(* IEC 61131-3 sources: AXOpen/src/components.cognex.vision/app/SystemConstants, 6 files *)

(* ---- plc_line_1518_HwIdentifiers.st ---- *)
CONFIGURATION HardwareIDs
    VAR_GLOBAL CONSTANT
        dm_280_HwID : UINT := UINT#299;
        dm_280_Acquisition_Control_Acquisition_Control_HwID : UINT := UINT#309;
        dm_280_Acquisition_Status_Acquisition_Status_HwID : UINT := UINT#306;
        dm_280_Rack_HwID : UINT := UINT#301;
        dm_280_Result_Data_128_bytes_Result_Data___128_bytes_HwID : UINT := UINT#303;
        dm_280_Results_Control_Results_Control_HwID : UINT := UINT#308;
        dm_280_Results_Status_Results_Status_HwID : UINT := UINT#305;
        dm_280_Soft_Event_Control_Soft_Event_Control_HwID : UINT := UINT#307;
        dm_280_User_Data_128_bytes_User_Data___128_bytes_HwID : UINT := UINT#304;
        dm_280_dm_280_HwID : UINT := UINT#302;
        dm_280_dm_280_DataMan_280_CC_B_HwID : UINT := UINT#310;
        dm_280_dm_280_profinet_HwID : UINT := UINT#298;
        dm_280_dm_280_profinet_Port_1_HwID : UINT := UINT#300;
        dm_300_HwID : UINT := UINT#286;
        dm_300_Acquisition_Control_Acquisition_Control_HwID : UINT := UINT#296;
        dm_300_Acquisition_Status_Acquisition_Status_HwID : UINT := UINT#293;
        dm_300_Rack_HwID : UINT := UINT#288;
        dm_300_Result_Data_64_bytes_Result_Data___64_bytes_HwID : UINT := UINT#290;
        dm_300_Results_Control_Results_Control_HwID : UINT := UINT#295;
        dm_300_Results_Status_Results_Status_HwID : UINT := UINT#292;
        dm_300_Soft_Event_Control_Soft_Event_Control_HwID : UINT := UINT#294;
        dm_300_User_Data_64_bytes_User_Data___64_bytes_HwID : UINT := UINT#291;
        dm_300_dm_300_HwID : UINT := UINT#289;
        dm_300_dm_300_DataMan_300_HwID : UINT := UINT#297;
        dm_300_dm_300_profinet_HwID : UINT := UINT#285;
        dm_300_dm_300_profinet_Port_1_HwID : UINT := UINT#287;
        is2800_HwID : UINT := UINT#258;
        is2800_Acquisition_Control_Acquisition_Control_HwID : UINT := UINT#269;
        is2800_Acquisition_Status_Acquisition_Status_HwID : UINT := UINT#264;
        is2800_Command_Control_Command_Control_HwID : UINT := UINT#266;
        is2800_Inspection_Control_Inspection_Control_HwID : UINT := UINT#268;
        is2800_Inspection_Status_Inspection_Status_HwID : UINT := UINT#265;
        is2800_Rack_HwID : UINT := UINT#260;
        is2800_Result_Data_64_bytes_Results___64_bytes_HwID : UINT := UINT#262;
        is2800_SoftEvent_Control_ExternalEvent_Control_HwID : UINT := UINT#267;
        is2800_User_Data_64_bytes_User_Data___64_bytes_HwID : UINT := UINT#263;
        is2800_is2800_HwID : UINT := UINT#261;
        is2800_is2800_In_Sight_IS28XX_CC_B_HwID : UINT := UINT#270;
        is2800_is2800_profinet_HwID : UINT := UINT#257;
        is2800_is2800_profinet_Port_1_HwID : UINT := UINT#259;
        is7600_HwID : UINT := UINT#272;
        is7600_Acquisition_Control_Acquisition_Control_HwID : UINT := UINT#283;
        is7600_Acquisition_Status_Acquisition_Status_HwID : UINT := UINT#279;
        is7600_Command_Control_Command_Control_HwID : UINT := UINT#280;
        is7600_Inspection_Control_Inspection_Control_HwID : UINT := UINT#282;
        is7600_Inspection_Status_Inspection_Status_HwID : UINT := UINT#278;
        is7600_Rack_HwID : UINT := UINT#274;
        is7600_Result_Data_64_bytes_Results___64_bytes_HwID : UINT := UINT#276;
        is7600_SoftEvent_Control_SoftEvent_Control_HwID : UINT := UINT#281;
        is7600_User_Data_64_bytes_User_Data___64_bytes_HwID : UINT := UINT#277;
        is7600_is7600_HwID : UINT := UINT#275;
        is7600_is7600_In_Sight_IS79XX_IS75XX_CC_B_HwID : UINT := UINT#284;
        is7600_is7600_profinet_HwID : UINT := UINT#271;
        is7600_is7600_profinet_Port_1_HwID : UINT := UINT#273;
        plc_line_1518_HwID : UINT := UINT#32;
        plc_line_1518_Rail_0_HwID : UINT := UINT#311;
        plc_line_1518_plc_line_1518_HwID : UINT := UINT#48;
        plc_line_1518_plc_line_1518_CPU_display_1_HwID : UINT := UINT#54;
        plc_line_1518_plc_line_1518_Card_reader_writer_1_HwID : UINT := UINT#51;
        plc_line_1518_plc_line_1518_OPC_UA_1_HwID : UINT := UINT#117;
        plc_line_1518_plc_line_1518_Virtual_communication_interface_HwID : UINT := UINT#135;
        plc_line_1518_plc_line_1518_profinet_x1_HwID : UINT := UINT#64;
        plc_line_1518_plc_line_1518_profinet_x1_Port_1_HwID : UINT := UINT#65;
        plc_line_1518_plc_line_1518_profinet_x1_Port_2_HwID : UINT := UINT#66;
        plc_line_1518_plc_line_1518_profinet_x2_HwID : UINT := UINT#72;
        plc_line_1518_plc_line_1518_profinet_x2_Port_3_HwID : UINT := UINT#73;
        plc_line_1518_plc_line_1518_profinet_x2_Port_4_HwID : UINT := UINT#74;
        plc_line_1518_plc_line_1518_profinet_x3_HwID : UINT := UINT#120;
        plc_line_1518_plc_line_1518_profinet_x3_Port_5_HwID : UINT := UINT#121;
        profinet_plc_line_1518_HwID : UINT := UINT#256;

    END_VAR
END_CONFIGURATION

(* ---- plc_line_1518_IoAddresses.st ---- *)
CONFIGURATION IoAddresses
    VAR_GLOBAL
        dm_280_Acquisition_Control_OutputAddress AT %QB343: BYTE;
        dm_280_Acquisition_Status_InputAddress_0 AT %IB373: BYTE;
        dm_280_Acquisition_Status_InputAddress_1 AT %IB374: BYTE;
        dm_280_Acquisition_Status_InputAddress_2 AT %IB375: BYTE;
        dm_280_Result_Data_128_bytes_InputAddress_0 AT %IL236: LWORD;
        dm_280_Result_Data_128_bytes_InputAddress_1 AT %IL244: LWORD;
        dm_280_Result_Data_128_bytes_InputAddress_2 AT %IL252: LWORD;
        dm_280_Result_Data_128_bytes_InputAddress_3 AT %IL260: LWORD;
        dm_280_Result_Data_128_bytes_InputAddress_4 AT %IL268: LWORD;
        dm_280_Result_Data_128_bytes_InputAddress_5 AT %IL276: LWORD;
        dm_280_Result_Data_128_bytes_InputAddress_6 AT %IL284: LWORD;
        dm_280_Result_Data_128_bytes_InputAddress_7 AT %IL292: LWORD;
        dm_280_Result_Data_128_bytes_InputAddress_8 AT %IL300: LWORD;
        dm_280_Result_Data_128_bytes_InputAddress_9 AT %IL308: LWORD;
        dm_280_Result_Data_128_bytes_InputAddress_10 AT %IL316: LWORD;
        dm_280_Result_Data_128_bytes_InputAddress_11 AT %IL324: LWORD;
        dm_280_Result_Data_128_bytes_InputAddress_12 AT %IL332: LWORD;
        dm_280_Result_Data_128_bytes_InputAddress_13 AT %IL340: LWORD;
        dm_280_Result_Data_128_bytes_InputAddress_14 AT %IL348: LWORD;
        dm_280_Result_Data_128_bytes_InputAddress_15 AT %IL356: LWORD;
        dm_280_Result_Data_128_bytes_InputAddress_16 AT %IL364: LWORD;
        dm_280_Results_Control_OutputAddress AT %QB342: BYTE;
        dm_280_Results_Status_InputAddress AT %IB372: BYTE;
        dm_280_Soft_Event_Control_InputAddress AT %IB376: BYTE;
        dm_280_Soft_Event_Control_OutputAddress AT %QB341: BYTE;
        dm_280_User_Data_128_bytes_OutputAddress_0 AT %QD209: DWORD;
        dm_280_User_Data_128_bytes_OutputAddress_1 AT %QD213: DWORD;
        dm_280_User_Data_128_bytes_OutputAddress_2 AT %QD217: DWORD;
        dm_280_User_Data_128_bytes_OutputAddress_3 AT %QD221: DWORD;
        dm_280_User_Data_128_bytes_OutputAddress_4 AT %QD225: DWORD;
        dm_280_User_Data_128_bytes_OutputAddress_5 AT %QD229: DWORD;
        dm_280_User_Data_128_bytes_OutputAddress_6 AT %QD233: DWORD;
        dm_280_User_Data_128_bytes_OutputAddress_7 AT %QD237: DWORD;
        dm_280_User_Data_128_bytes_OutputAddress_8 AT %QD241: DWORD;
        dm_280_User_Data_128_bytes_OutputAddress_9 AT %QD245: DWORD;
        dm_280_User_Data_128_bytes_OutputAddress_10 AT %QD249: DWORD;
        dm_280_User_Data_128_bytes_OutputAddress_11 AT %QD253: DWORD;
        dm_280_User_Data_128_bytes_OutputAddress_12 AT %QD257: DWORD;
        dm_280_User_Data_128_bytes_OutputAddress_13 AT %QD261: DWORD;
        dm_280_User_Data_128_bytes_OutputAddress_14 AT %QD265: DWORD;
        dm_280_User_Data_128_bytes_OutputAddress_15 AT %QD269: DWORD;
        dm_280_User_Data_128_bytes_OutputAddress_16 AT %QD273: DWORD;
        dm_280_User_Data_128_bytes_OutputAddress_17 AT %QD277: DWORD;
        dm_280_User_Data_128_bytes_OutputAddress_18 AT %QD281: DWORD;
        dm_280_User_Data_128_bytes_OutputAddress_19 AT %QD285: DWORD;
        dm_280_User_Data_128_bytes_OutputAddress_20 AT %QD289: DWORD;
        dm_280_User_Data_128_bytes_OutputAddress_21 AT %QD293: DWORD;
        dm_280_User_Data_128_bytes_OutputAddress_22 AT %QD297: DWORD;
        dm_280_User_Data_128_bytes_OutputAddress_23 AT %QD301: DWORD;
        dm_280_User_Data_128_bytes_OutputAddress_24 AT %QD305: DWORD;
        dm_280_User_Data_128_bytes_OutputAddress_25 AT %QD309: DWORD;
        dm_280_User_Data_128_bytes_OutputAddress_26 AT %QD313: DWORD;
        dm_280_User_Data_128_bytes_OutputAddress_27 AT %QD317: DWORD;
        dm_280_User_Data_128_bytes_OutputAddress_28 AT %QD321: DWORD;
        dm_280_User_Data_128_bytes_OutputAddress_29 AT %QD325: DWORD;
        dm_280_User_Data_128_bytes_OutputAddress_30 AT %QD329: DWORD;
        dm_280_User_Data_128_bytes_OutputAddress_31 AT %QD333: DWORD;
        dm_280_User_Data_128_bytes_OutputAddress_32 AT %QD337: DWORD;
        dm_300_Acquisition_Control_OutputAddress AT %QB208: BYTE;
        dm_300_Acquisition_Status_InputAddress_0 AT %IB232: BYTE;
        dm_300_Acquisition_Status_InputAddress_1 AT %IB233: BYTE;
        dm_300_Acquisition_Status_InputAddress_2 AT %IB234: BYTE;
        dm_300_Result_Data_64_bytes_InputAddress_0 AT %IL159: LWORD;
        dm_300_Result_Data_64_bytes_InputAddress_1 AT %IL167: LWORD;
        dm_300_Result_Data_64_bytes_InputAddress_2 AT %IL175: LWORD;
        dm_300_Result_Data_64_bytes_InputAddress_3 AT %IL183: LWORD;
        dm_300_Result_Data_64_bytes_InputAddress_4 AT %IL191: LWORD;
        dm_300_Result_Data_64_bytes_InputAddress_5 AT %IL199: LWORD;
        dm_300_Result_Data_64_bytes_InputAddress_6 AT %IL207: LWORD;
        dm_300_Result_Data_64_bytes_InputAddress_7 AT %IL215: LWORD;
        dm_300_Result_Data_64_bytes_InputAddress_8 AT %IL223: LWORD;
        dm_300_Results_Control_OutputAddress AT %QB207: BYTE;
        dm_300_Results_Status_InputAddress AT %IB231: BYTE;
        dm_300_Soft_Event_Control_InputAddress AT %IB235: BYTE;
        dm_300_Soft_Event_Control_OutputAddress AT %QB206: BYTE;
        dm_300_User_Data_64_bytes_OutputAddress_0 AT %QD138: DWORD;
        dm_300_User_Data_64_bytes_OutputAddress_1 AT %QD142: DWORD;
        dm_300_User_Data_64_bytes_OutputAddress_2 AT %QD146: DWORD;
        dm_300_User_Data_64_bytes_OutputAddress_3 AT %QD150: DWORD;
        dm_300_User_Data_64_bytes_OutputAddress_4 AT %QD154: DWORD;
        dm_300_User_Data_64_bytes_OutputAddress_5 AT %QD158: DWORD;
        dm_300_User_Data_64_bytes_OutputAddress_6 AT %QD162: DWORD;
        dm_300_User_Data_64_bytes_OutputAddress_7 AT %QD166: DWORD;
        dm_300_User_Data_64_bytes_OutputAddress_8 AT %QD170: DWORD;
        dm_300_User_Data_64_bytes_OutputAddress_9 AT %QD174: DWORD;
        dm_300_User_Data_64_bytes_OutputAddress_10 AT %QD178: DWORD;
        dm_300_User_Data_64_bytes_OutputAddress_11 AT %QD182: DWORD;
        dm_300_User_Data_64_bytes_OutputAddress_12 AT %QD186: DWORD;
        dm_300_User_Data_64_bytes_OutputAddress_13 AT %QD190: DWORD;
        dm_300_User_Data_64_bytes_OutputAddress_14 AT %QD194: DWORD;
        dm_300_User_Data_64_bytes_OutputAddress_15 AT %QD198: DWORD;
        dm_300_User_Data_64_bytes_OutputAddress_16 AT %QD202: DWORD;
        is2800_Acquisition_Control_OutputAddress AT %QB68: BYTE;
        is2800_Acquisition_Status_InputAddress AT %ID68: DWORD;
        is2800_Command_Control_InputAddress AT %ID76: DWORD;
        is2800_Command_Control_OutputAddress AT %QW64: WORD;
        is2800_Inspection_Control_OutputAddress AT %QB67: BYTE;
        is2800_Inspection_Status_InputAddress AT %ID72: DWORD;
        is2800_Result_Data_64_bytes_InputAddress_0 AT %ID0: DWORD;
        is2800_Result_Data_64_bytes_InputAddress_1 AT %ID4: DWORD;
        is2800_Result_Data_64_bytes_InputAddress_2 AT %ID8: DWORD;
        is2800_Result_Data_64_bytes_InputAddress_3 AT %ID12: DWORD;
        is2800_Result_Data_64_bytes_InputAddress_4 AT %ID16: DWORD;
        is2800_Result_Data_64_bytes_InputAddress_5 AT %ID20: DWORD;
        is2800_Result_Data_64_bytes_InputAddress_6 AT %ID24: DWORD;
        is2800_Result_Data_64_bytes_InputAddress_7 AT %ID28: DWORD;
        is2800_Result_Data_64_bytes_InputAddress_8 AT %ID32: DWORD;
        is2800_Result_Data_64_bytes_InputAddress_9 AT %ID36: DWORD;
        is2800_Result_Data_64_bytes_InputAddress_10 AT %ID40: DWORD;
        is2800_Result_Data_64_bytes_InputAddress_11 AT %ID44: DWORD;
        is2800_Result_Data_64_bytes_InputAddress_12 AT %ID48: DWORD;
        is2800_Result_Data_64_bytes_InputAddress_13 AT %ID52: DWORD;
        is2800_Result_Data_64_bytes_InputAddress_14 AT %ID56: DWORD;
        is2800_Result_Data_64_bytes_InputAddress_15 AT %ID60: DWORD;
        is2800_Result_Data_64_bytes_InputAddress_16 AT %ID64: DWORD;
        is2800_SoftEvent_Control_InputAddress AT %IB80: BYTE;
        is2800_SoftEvent_Control_OutputAddress AT %QB66: BYTE;
        is2800_User_Data_64_bytes_OutputAddress_0 AT %QL0: LWORD;
        is2800_User_Data_64_bytes_OutputAddress_1 AT %QL8: LWORD;
        is2800_User_Data_64_bytes_OutputAddress_2 AT %QL16: LWORD;
        is2800_User_Data_64_bytes_OutputAddress_3 AT %QL24: LWORD;
        is2800_User_Data_64_bytes_OutputAddress_4 AT %QL32: LWORD;
        is2800_User_Data_64_bytes_OutputAddress_5 AT %QL40: LWORD;
        is2800_User_Data_64_bytes_OutputAddress_6 AT %QL48: LWORD;
        is2800_User_Data_64_bytes_OutputAddress_7 AT %QL56: LWORD;
        is7600_Acquisition_Control_OutputAddress AT %QB137: BYTE;
        is7600_Acquisition_Status_InputAddress_0 AT %IB153: BYTE;
        is7600_Acquisition_Status_InputAddress_1 AT %IB154: BYTE;
        is7600_Acquisition_Status_InputAddress_2 AT %IB155: BYTE;
        is7600_Command_Control_InputAddress AT %IW156: WORD;
        is7600_Command_Control_OutputAddress AT %QW133: WORD;
        is7600_Inspection_Control_OutputAddress AT %QB136: BYTE;
        is7600_Inspection_Status_InputAddress AT %ID149: DWORD;
        is7600_Result_Data_64_bytes_InputAddress_0 AT %ID81: DWORD;
        is7600_Result_Data_64_bytes_InputAddress_1 AT %ID85: DWORD;
        is7600_Result_Data_64_bytes_InputAddress_2 AT %ID89: DWORD;
        is7600_Result_Data_64_bytes_InputAddress_3 AT %ID93: DWORD;
        is7600_Result_Data_64_bytes_InputAddress_4 AT %ID97: DWORD;
        is7600_Result_Data_64_bytes_InputAddress_5 AT %ID101: DWORD;
        is7600_Result_Data_64_bytes_InputAddress_6 AT %ID105: DWORD;
        is7600_Result_Data_64_bytes_InputAddress_7 AT %ID109: DWORD;
        is7600_Result_Data_64_bytes_InputAddress_8 AT %ID113: DWORD;
        is7600_Result_Data_64_bytes_InputAddress_9 AT %ID117: DWORD;
        is7600_Result_Data_64_bytes_InputAddress_10 AT %ID121: DWORD;
        is7600_Result_Data_64_bytes_InputAddress_11 AT %ID125: DWORD;
        is7600_Result_Data_64_bytes_InputAddress_12 AT %ID129: DWORD;
        is7600_Result_Data_64_bytes_InputAddress_13 AT %ID133: DWORD;
        is7600_Result_Data_64_bytes_InputAddress_14 AT %ID137: DWORD;
        is7600_Result_Data_64_bytes_InputAddress_15 AT %ID141: DWORD;
        is7600_Result_Data_64_bytes_InputAddress_16 AT %ID145: DWORD;
        is7600_SoftEvent_Control_InputAddress AT %IB158: BYTE;
        is7600_SoftEvent_Control_OutputAddress AT %QB135: BYTE;
        is7600_User_Data_64_bytes_OutputAddress_0 AT %QL69: LWORD;
        is7600_User_Data_64_bytes_OutputAddress_1 AT %QL77: LWORD;
        is7600_User_Data_64_bytes_OutputAddress_2 AT %QL85: LWORD;
        is7600_User_Data_64_bytes_OutputAddress_3 AT %QL93: LWORD;
        is7600_User_Data_64_bytes_OutputAddress_4 AT %QL101: LWORD;
        is7600_User_Data_64_bytes_OutputAddress_5 AT %QL109: LWORD;
        is7600_User_Data_64_bytes_OutputAddress_6 AT %QL117: LWORD;
        is7600_User_Data_64_bytes_OutputAddress_7 AT %QL125: LWORD;

    END_VAR
END_CONFIGURATION

(* ---- plc_line_HwIdentifiers.st ---- *)
CONFIGURATION HardwareIDs
    VAR_GLOBAL CONSTANT
        is7600_HwID : UINT := UINT#259;
        is7600_Acquisition_Control_Acquisition_Control_HwID : UINT := UINT#269;
        is7600_Acquisition_Status_Acquisition_Status_HwID : UINT := UINT#265;
        is7600_Command_Control_Command_Control_HwID : UINT := UINT#266;
        is7600_Inspection_Control_Inspection_Control_HwID : UINT := UINT#268;
        is7600_Inspection_Status_Inspection_Status_HwID : UINT := UINT#264;
        is7600_Rack_HwID : UINT := UINT#260;
        is7600_Result_Data_64_bytes_Results___64_bytes_HwID : UINT := UINT#262;
        is7600_SoftEvent_Control_SoftEvent_Control_HwID : UINT := UINT#267;
        is7600_User_Data_64_bytes_User_Data___64_bytes_HwID : UINT := UINT#263;
        is7600_is7600_HwID : UINT := UINT#261;
        is7600_is7600_In_Sight_IS79XX_IS75XX_CC_B_HwID : UINT := UINT#270;
        is7600_is7600_profinet_HwID : UINT := UINT#257;
        is7600_is7600_profinet_Port_1_HwID : UINT := UINT#258;
        plc_line_HwID : UINT := UINT#32;
        plc_line_Rail_0_HwID : UINT := UINT#297;
        plc_line_plc_line_HwID : UINT := UINT#48;
        plc_line_plc_line_CPU_display_1_HwID : UINT := UINT#54;
        plc_line_plc_line_Card_reader_writer_1_HwID : UINT := UINT#51;
        plc_line_plc_line_DP_interface_1_HwID : UINT := UINT#60;
        plc_line_plc_line_OPC_UA_1_HwID : UINT := UINT#117;
        plc_line_plc_line_profinet_x1_HwID : UINT := UINT#64;
        plc_line_plc_line_profinet_x1_Port_1_HwID : UINT := UINT#65;
        plc_line_plc_line_profinet_x1_Port_2_HwID : UINT := UINT#66;
        plc_line_plc_line_profinet_x2_HwID : UINT := UINT#72;
        plc_line_plc_line_profinet_x2_Port_3_HwID : UINT := UINT#73;
        plc_line_plc_line_virtual_communication_interface_HwID : UINT := UINT#135;
        profinet_plc_line_HwID : UINT := UINT#256;
        reader_st1_HwID : UINT := UINT#286;
        reader_st1_Acquisition_Control_Acquisition_Control_HwID : UINT := UINT#295;
        reader_st1_Acquisition_Status_Acquisition_Status_HwID : UINT := UINT#292;
        reader_st1_Rack_HwID : UINT := UINT#287;
        reader_st1_Result_Data_128_bytes_Result_Data___128_bytes_HwID : UINT := UINT#289;
        reader_st1_Results_Control_Results_Control_HwID : UINT := UINT#294;
        reader_st1_Results_Status_Results_Status_HwID : UINT := UINT#291;
        reader_st1_Soft_Event_Control_Soft_Event_Control_HwID : UINT := UINT#293;
        reader_st1_User_Data_128_bytes_User_Data___128_bytes_HwID : UINT := UINT#290;
        reader_st1_reader_st1_HwID : UINT := UINT#288;
        reader_st1_reader_st1_DataMan_280_CC_B_HwID : UINT := UINT#296;
        reader_st1_reader_st1_profinet_HwID : UINT := UINT#284;
        reader_st1_reader_st1_profinet_Port_1_HwID : UINT := UINT#285;
        reader_st2_HwID : UINT := UINT#273;
        reader_st2_Acquisition_Control_Acquisition_Control_HwID : UINT := UINT#282;
        reader_st2_Acquisition_Status_Acquisition_Status_HwID : UINT := UINT#279;
        reader_st2_Rack_HwID : UINT := UINT#274;
        reader_st2_Result_Data_64_bytes_Result_Data___64_bytes_HwID : UINT := UINT#276;
        reader_st2_Results_Control_Results_Control_HwID : UINT := UINT#281;
        reader_st2_Results_Status_Results_Status_HwID : UINT := UINT#278;
        reader_st2_Soft_Event_Control_Soft_Event_Control_HwID : UINT := UINT#280;
        reader_st2_User_Data_64_bytes_User_Data___64_bytes_HwID : UINT := UINT#277;
        reader_st2_reader_st2_HwID : UINT := UINT#275;
        reader_st2_reader_st2_DataMan_300_HwID : UINT := UINT#283;
        reader_st2_reader_st2_profinet_HwID : UINT := UINT#271;
        reader_st2_reader_st2_profinet_Port_1_HwID : UINT := UINT#272;

    END_VAR
END_CONFIGURATION

(* ---- plc_line_IoAddresses.st ---- *)
CONFIGURATION IoAddresses
    VAR_GLOBAL
        is7600_Acquisition_Control_OutputAddress AT %QB68: BYTE;
        is7600_Acquisition_Status_InputAddress_0 AT %IB72: BYTE;
        is7600_Acquisition_Status_InputAddress_1 AT %IB73: BYTE;
        is7600_Acquisition_Status_InputAddress_2 AT %IB74: BYTE;
        is7600_Command_Control_InputAddress AT %IW75: WORD;
        is7600_Command_Control_OutputAddress AT %QW64: WORD;
        is7600_Inspection_Control_OutputAddress AT %QB67: BYTE;
        is7600_Inspection_Status_InputAddress AT %ID68: DWORD;
        is7600_Result_Data_64_bytes_InputAddress_0 AT %ID0: DWORD;
        is7600_Result_Data_64_bytes_InputAddress_1 AT %ID4: DWORD;
        is7600_Result_Data_64_bytes_InputAddress_2 AT %ID8: DWORD;
        is7600_Result_Data_64_bytes_InputAddress_3 AT %ID12: DWORD;
        is7600_Result_Data_64_bytes_InputAddress_4 AT %ID16: DWORD;
        is7600_Result_Data_64_bytes_InputAddress_5 AT %ID20: DWORD;
        is7600_Result_Data_64_bytes_InputAddress_6 AT %ID24: DWORD;
        is7600_Result_Data_64_bytes_InputAddress_7 AT %ID28: DWORD;
        is7600_Result_Data_64_bytes_InputAddress_8 AT %ID32: DWORD;
        is7600_Result_Data_64_bytes_InputAddress_9 AT %ID36: DWORD;
        is7600_Result_Data_64_bytes_InputAddress_10 AT %ID40: DWORD;
        is7600_Result_Data_64_bytes_InputAddress_11 AT %ID44: DWORD;
        is7600_Result_Data_64_bytes_InputAddress_12 AT %ID48: DWORD;
        is7600_Result_Data_64_bytes_InputAddress_13 AT %ID52: DWORD;
        is7600_Result_Data_64_bytes_InputAddress_14 AT %ID56: DWORD;
        is7600_Result_Data_64_bytes_InputAddress_15 AT %ID60: DWORD;
        is7600_Result_Data_64_bytes_InputAddress_16 AT %ID64: DWORD;
        is7600_SoftEvent_Control_InputAddress AT %IB77: BYTE;
        is7600_SoftEvent_Control_OutputAddress AT %QB66: BYTE;
        is7600_User_Data_64_bytes_OutputAddress_0 AT %QL0: LWORD;
        is7600_User_Data_64_bytes_OutputAddress_1 AT %QL8: LWORD;
        is7600_User_Data_64_bytes_OutputAddress_2 AT %QL16: LWORD;
        is7600_User_Data_64_bytes_OutputAddress_3 AT %QL24: LWORD;
        is7600_User_Data_64_bytes_OutputAddress_4 AT %QL32: LWORD;
        is7600_User_Data_64_bytes_OutputAddress_5 AT %QL40: LWORD;
        is7600_User_Data_64_bytes_OutputAddress_6 AT %QL48: LWORD;
        is7600_User_Data_64_bytes_OutputAddress_7 AT %QL56: LWORD;
        reader_st1_Acquisition_Control_OutputAddress AT %QB274: BYTE;
        reader_st1_Acquisition_Status_InputAddress_0 AT %IB293: BYTE;
        reader_st1_Acquisition_Status_InputAddress_1 AT %IB294: BYTE;
        reader_st1_Acquisition_Status_InputAddress_2 AT %IB295: BYTE;
        reader_st1_Result_Data_128_bytes_InputAddress_0 AT %IL155: LWORD;
        reader_st1_Result_Data_128_bytes_InputAddress_1 AT %IL163: LWORD;
        reader_st1_Result_Data_128_bytes_InputAddress_2 AT %IL171: LWORD;
        reader_st1_Result_Data_128_bytes_InputAddress_3 AT %IL179: LWORD;
        reader_st1_Result_Data_128_bytes_InputAddress_4 AT %IL187: LWORD;
        reader_st1_Result_Data_128_bytes_InputAddress_5 AT %IL195: LWORD;
        reader_st1_Result_Data_128_bytes_InputAddress_6 AT %IL203: LWORD;
        reader_st1_Result_Data_128_bytes_InputAddress_7 AT %IL211: LWORD;
        reader_st1_Result_Data_128_bytes_InputAddress_8 AT %IL219: LWORD;
        reader_st1_Result_Data_128_bytes_InputAddress_9 AT %IL227: LWORD;
        reader_st1_Result_Data_128_bytes_InputAddress_10 AT %IL235: LWORD;
        reader_st1_Result_Data_128_bytes_InputAddress_11 AT %IL243: LWORD;
        reader_st1_Result_Data_128_bytes_InputAddress_12 AT %IL251: LWORD;
        reader_st1_Result_Data_128_bytes_InputAddress_13 AT %IL259: LWORD;
        reader_st1_Result_Data_128_bytes_InputAddress_14 AT %IL267: LWORD;
        reader_st1_Result_Data_128_bytes_InputAddress_15 AT %IL275: LWORD;
        reader_st1_Result_Data_128_bytes_InputAddress_16 AT %IL283: LWORD;
        reader_st1_Results_Control_OutputAddress AT %QB273: BYTE;
        reader_st1_Results_Status_InputAddress AT %IB292: BYTE;
        reader_st1_Soft_Event_Control_InputAddress AT %IB291: BYTE;
        reader_st1_Soft_Event_Control_OutputAddress AT %QB272: BYTE;
        reader_st1_User_Data_128_bytes_OutputAddress_0 AT %QD140: DWORD;
        reader_st1_User_Data_128_bytes_OutputAddress_1 AT %QD144: DWORD;
        reader_st1_User_Data_128_bytes_OutputAddress_2 AT %QD148: DWORD;
        reader_st1_User_Data_128_bytes_OutputAddress_3 AT %QD152: DWORD;
        reader_st1_User_Data_128_bytes_OutputAddress_4 AT %QD156: DWORD;
        reader_st1_User_Data_128_bytes_OutputAddress_5 AT %QD160: DWORD;
        reader_st1_User_Data_128_bytes_OutputAddress_6 AT %QD164: DWORD;
        reader_st1_User_Data_128_bytes_OutputAddress_7 AT %QD168: DWORD;
        reader_st1_User_Data_128_bytes_OutputAddress_8 AT %QD172: DWORD;
        reader_st1_User_Data_128_bytes_OutputAddress_9 AT %QD176: DWORD;
        reader_st1_User_Data_128_bytes_OutputAddress_10 AT %QD180: DWORD;
        reader_st1_User_Data_128_bytes_OutputAddress_11 AT %QD184: DWORD;
        reader_st1_User_Data_128_bytes_OutputAddress_12 AT %QD188: DWORD;
        reader_st1_User_Data_128_bytes_OutputAddress_13 AT %QD192: DWORD;
        reader_st1_User_Data_128_bytes_OutputAddress_14 AT %QD196: DWORD;
        reader_st1_User_Data_128_bytes_OutputAddress_15 AT %QD200: DWORD;
        reader_st1_User_Data_128_bytes_OutputAddress_16 AT %QD204: DWORD;
        reader_st1_User_Data_128_bytes_OutputAddress_17 AT %QD208: DWORD;
        reader_st1_User_Data_128_bytes_OutputAddress_18 AT %QD212: DWORD;
        reader_st1_User_Data_128_bytes_OutputAddress_19 AT %QD216: DWORD;
        reader_st1_User_Data_128_bytes_OutputAddress_20 AT %QD220: DWORD;
        reader_st1_User_Data_128_bytes_OutputAddress_21 AT %QD224: DWORD;
        reader_st1_User_Data_128_bytes_OutputAddress_22 AT %QD228: DWORD;
        reader_st1_User_Data_128_bytes_OutputAddress_23 AT %QD232: DWORD;
        reader_st1_User_Data_128_bytes_OutputAddress_24 AT %QD236: DWORD;
        reader_st1_User_Data_128_bytes_OutputAddress_25 AT %QD240: DWORD;
        reader_st1_User_Data_128_bytes_OutputAddress_26 AT %QD244: DWORD;
        reader_st1_User_Data_128_bytes_OutputAddress_27 AT %QD248: DWORD;
        reader_st1_User_Data_128_bytes_OutputAddress_28 AT %QD252: DWORD;
        reader_st1_User_Data_128_bytes_OutputAddress_29 AT %QD256: DWORD;
        reader_st1_User_Data_128_bytes_OutputAddress_30 AT %QD260: DWORD;
        reader_st1_User_Data_128_bytes_OutputAddress_31 AT %QD264: DWORD;
        reader_st1_User_Data_128_bytes_OutputAddress_32 AT %QD268: DWORD;
        reader_st2_Acquisition_Control_OutputAddress AT %QB139: BYTE;
        reader_st2_Acquisition_Status_InputAddress_0 AT %IB152: BYTE;
        reader_st2_Acquisition_Status_InputAddress_1 AT %IB153: BYTE;
        reader_st2_Acquisition_Status_InputAddress_2 AT %IB154: BYTE;
        reader_st2_Result_Data_64_bytes_InputAddress_0 AT %IL78: LWORD;
        reader_st2_Result_Data_64_bytes_InputAddress_1 AT %IL86: LWORD;
        reader_st2_Result_Data_64_bytes_InputAddress_2 AT %IL94: LWORD;
        reader_st2_Result_Data_64_bytes_InputAddress_3 AT %IL102: LWORD;
        reader_st2_Result_Data_64_bytes_InputAddress_4 AT %IL110: LWORD;
        reader_st2_Result_Data_64_bytes_InputAddress_5 AT %IL118: LWORD;
        reader_st2_Result_Data_64_bytes_InputAddress_6 AT %IL126: LWORD;
        reader_st2_Result_Data_64_bytes_InputAddress_7 AT %IL134: LWORD;
        reader_st2_Result_Data_64_bytes_InputAddress_8 AT %IL142: LWORD;
        reader_st2_Results_Control_OutputAddress AT %QB138: BYTE;
        reader_st2_Results_Status_InputAddress AT %IB151: BYTE;
        reader_st2_Soft_Event_Control_InputAddress AT %IB150: BYTE;
        reader_st2_Soft_Event_Control_OutputAddress AT %QB137: BYTE;
        reader_st2_User_Data_64_bytes_OutputAddress_0 AT %QD69: DWORD;
        reader_st2_User_Data_64_bytes_OutputAddress_1 AT %QD73: DWORD;
        reader_st2_User_Data_64_bytes_OutputAddress_2 AT %QD77: DWORD;
        reader_st2_User_Data_64_bytes_OutputAddress_3 AT %QD81: DWORD;
        reader_st2_User_Data_64_bytes_OutputAddress_4 AT %QD85: DWORD;
        reader_st2_User_Data_64_bytes_OutputAddress_5 AT %QD89: DWORD;
        reader_st2_User_Data_64_bytes_OutputAddress_6 AT %QD93: DWORD;
        reader_st2_User_Data_64_bytes_OutputAddress_7 AT %QD97: DWORD;
        reader_st2_User_Data_64_bytes_OutputAddress_8 AT %QD101: DWORD;
        reader_st2_User_Data_64_bytes_OutputAddress_9 AT %QD105: DWORD;
        reader_st2_User_Data_64_bytes_OutputAddress_10 AT %QD109: DWORD;
        reader_st2_User_Data_64_bytes_OutputAddress_11 AT %QD113: DWORD;
        reader_st2_User_Data_64_bytes_OutputAddress_12 AT %QD117: DWORD;
        reader_st2_User_Data_64_bytes_OutputAddress_13 AT %QD121: DWORD;
        reader_st2_User_Data_64_bytes_OutputAddress_14 AT %QD125: DWORD;
        reader_st2_User_Data_64_bytes_OutputAddress_15 AT %QD129: DWORD;
        reader_st2_User_Data_64_bytes_OutputAddress_16 AT %QD133: DWORD;

    END_VAR
END_CONFIGURATION

(* ---- plc_main_HwIdentifiers.st ---- *)
CONFIGURATION HardwareIDs
    VAR_GLOBAL CONSTANT
        CommunicationCard_HwID : UINT := UINT#258;
        CommunicationCard_CommunicationCard_HwID : UINT := UINT#261;
        CommunicationCard_CommunicationCard_Communication_Card_CC24_HwID : UINT := UINT#279;
        CommunicationCard_CommunicationCard_profinet_HwID : UINT := UINT#257;
        CommunicationCard_CommunicationCard_profinet_Port_1_HwID : UINT := UINT#259;
        CommunicationCard_Engine_Control_1_Engine_Control_HwID : UINT := UINT#277;
        CommunicationCard_Engine_Control_2_Engine_Control_HwID : UINT := UINT#276;
        CommunicationCard_Engine_Control_3_Engine_Control_HwID : UINT := UINT#275;
        CommunicationCard_Engine_Control_4_Engine_Control_HwID : UINT := UINT#274;
        CommunicationCard_Rack_HwID : UINT := UINT#260;
        CommunicationCard_Result_Data_240_bytes_1_Results___240_bytes_HwID : UINT := UINT#272;
        CommunicationCard_Result_Data_240_bytes_2_Results___240_bytes_HwID : UINT := UINT#266;
        CommunicationCard_Result_Data_240_bytes_3_Results___240_bytes_HwID : UINT := UINT#265;
        CommunicationCard_Result_Data_240_bytes_4_Results___240_bytes_HwID : UINT := UINT#264;
        CommunicationCard_Result_Data_240_bytes_5_Results___240_bytes_HwID : UINT := UINT#263;
        CommunicationCard_Result_Data_64_bytes_1_Results___64_bytes_HwID : UINT := UINT#262;
        CommunicationCard_System_Control_System_Control_HwID : UINT := UINT#278;
        CommunicationCard_User_Data_240_bytes_1_User_Data___240_bytes_HwID : UINT := UINT#273;
        CommunicationCard_User_Data_240_bytes_2_User_Data___240_bytes_HwID : UINT := UINT#271;
        CommunicationCard_User_Data_240_bytes_3_User_Data___240_bytes_HwID : UINT := UINT#270;
        CommunicationCard_User_Data_240_bytes_4_User_Data___240_bytes_HwID : UINT := UINT#269;
        CommunicationCard_User_Data_240_bytes_5_User_Data___240_bytes_HwID : UINT := UINT#268;
        CommunicationCard_User_Data_64_bytes_1_User_Data___64_bytes_HwID : UINT := UINT#267;
        plc_main_HwID : UINT := UINT#32;
        plc_main_Rail_0_HwID : UINT := UINT#327;
        plc_main_plc_main_HwID : UINT := UINT#48;
        plc_main_plc_main_CPU_display_1_HwID : UINT := UINT#54;
        plc_main_plc_main_Card_reader_writer_1_HwID : UINT := UINT#51;
        plc_main_plc_main_OPC_UA_1_HwID : UINT := UINT#117;
        plc_main_plc_main_Virtual_communication_interface_HwID : UINT := UINT#135;
        plc_main_plc_main_profinet_x1_HwID : UINT := UINT#64;
        plc_main_plc_main_profinet_x1_Port_1_HwID : UINT := UINT#65;
        plc_main_plc_main_profinet_x1_Port_2_HwID : UINT := UINT#66;
        plc_main_plc_main_profinet_x2_HwID : UINT := UINT#72;
        plc_main_plc_main_profinet_x2_Port_3_HwID : UINT := UINT#73;
        plc_main_plc_main_profinet_x2_Port_4_HwID : UINT := UINT#74;
        plc_main_plc_main_profinet_x3_HwID : UINT := UINT#120;
        plc_main_plc_main_profinet_x3_Port_5_HwID : UINT := UINT#121;
        profinet_plc_main_HwID : UINT := UINT#256;
        st10_dm280_HwID : UINT := UINT#295;
        st10_dm280_Acquisition_Control_Acquisition_Control_HwID : UINT := UINT#305;
        st10_dm280_Acquisition_Status_Acquisition_Status_HwID : UINT := UINT#302;
        st10_dm280_Rack_HwID : UINT := UINT#297;
        st10_dm280_Result_Data_128_bytes_Result_Data___128_bytes_HwID : UINT := UINT#299;
        st10_dm280_Results_Control_Results_Control_HwID : UINT := UINT#304;
        st10_dm280_Results_Status_Results_Status_HwID : UINT := UINT#301;
        st10_dm280_Soft_Event_Control_Soft_Event_Control_HwID : UINT := UINT#303;
        st10_dm280_User_Data_128_bytes_User_Data___128_bytes_HwID : UINT := UINT#300;
        st10_dm280_st10_dm280_HwID : UINT := UINT#298;
        st10_dm280_st10_dm280_DataMan_280_CC_B_HwID : UINT := UINT#306;
        st10_dm280_st10_dm280_profinet_HwID : UINT := UINT#294;
        st10_dm280_st10_dm280_profinet_Port_1_HwID : UINT := UINT#296;
        st10_is2802m_HwID : UINT := UINT#308;
        st10_is2802m_Acquisition_Control_Acquisition_Control_HwID : UINT := UINT#325;
        st10_is2802m_Acquisition_Status_Acquisition_Status_HwID : UINT := UINT#320;
        st10_is2802m_Command_Control_Command_Control_HwID : UINT := UINT#322;
        st10_is2802m_Inspection_Control_Inspection_Control_HwID : UINT := UINT#324;
        st10_is2802m_Inspection_Status_Inspection_Status_HwID : UINT := UINT#321;
        st10_is2802m_Rack_HwID : UINT := UINT#310;
        st10_is2802m_Result_Data_250_bytes_1_Results___250_bytes_HwID : UINT := UINT#315;
        st10_is2802m_Result_Data_250_bytes_2_Results___250_bytes_HwID : UINT := UINT#314;
        st10_is2802m_Result_Data_250_bytes_3_Results___250_bytes_HwID : UINT := UINT#313;
        st10_is2802m_Result_Data_250_bytes_4_Results___250_bytes_HwID : UINT := UINT#312;
        st10_is2802m_SoftEvent_Control_ExternalEvent_Control_HwID : UINT := UINT#323;
        st10_is2802m_User_Data_254_bytes_1_User_Data___254_bytes_HwID : UINT := UINT#319;
        st10_is2802m_User_Data_254_bytes_2_User_Data___254_bytes_HwID : UINT := UINT#318;
        st10_is2802m_User_Data_254_bytes_3_User_Data___254_bytes_HwID : UINT := UINT#317;
        st10_is2802m_User_Data_254_bytes_4_User_Data___254_bytes_HwID : UINT := UINT#316;
        st10_is2802m_st10_is2802m_HwID : UINT := UINT#311;
        st10_is2802m_st10_is2802m_In_Sight_IS28XX_CC_B_HwID : UINT := UINT#326;
        st10_is2802m_st10_is2802m_profinet_HwID : UINT := UINT#307;
        st10_is2802m_st10_is2802m_profinet_Port_1_HwID : UINT := UINT#309;
        st20_is2000_navigation_HwID : UINT := UINT#281;
        st20_is2000_navigation_Acquisition_Control_Acquisition_Control_HwID : UINT := UINT#292;
        st20_is2000_navigation_Acquisition_Status_Acquisition_Status_HwID : UINT := UINT#288;
        st20_is2000_navigation_Command_Control_Command_Control_HwID : UINT := UINT#289;
        st20_is2000_navigation_Inspection_Control_Inspection_Control_HwID : UINT := UINT#291;
        st20_is2000_navigation_Inspection_Status_Inspection_Status_HwID : UINT := UINT#287;
        st20_is2000_navigation_Rack_HwID : UINT := UINT#283;
        st20_is2000_navigation_Result_Data_64_bytes_Results___64_bytes_HwID : UINT := UINT#285;
        st20_is2000_navigation_SoftEvent_Control_SoftEvent_Control_HwID : UINT := UINT#290;
        st20_is2000_navigation_User_Data_64_bytes_User_Data___64_bytes_HwID : UINT := UINT#286;
        st20_is2000_navigation_st20_is2000_navigation_HwID : UINT := UINT#284;
        st20_is2000_navigation_st20_is2000_navigation_In_Sight_IS2XXX_CC_B_HwID : UINT := UINT#293;
        st20_is2000_navigation_st20_is2000_navigation_profinet_HwID : UINT := UINT#280;
        st20_is2000_navigation_st20_is2000_navigation_profinet_Port_1_HwID : UINT := UINT#282;

    END_VAR
END_CONFIGURATION
